TYPE ST_Recipe :
	STRUCT
		LiftPosition_Up	  : LREAL := 100;
		LiftPosition_Down : LREAL := 0;
	END_STRUCT
END_TYPE

(* stored: Version 1.1.0.1
   DUT ST_Recipe: Id {5ad52013-de8a-4f34-9327-e4b2e37f9d37} *)
